// TIA Portal V17 export
// export: Created 2023-04-03T06:31:28.7566362Z, ExportSetting WithDefaults, DisplayName Totally Integrated Automation Portal, DisplayVersion V17 Update 4, DisplayName TIA Portal Openness, DisplayVersion V17 Update 4, DisplayName TIA Portal Version Control Interface, DisplayVersion V17, DisplayName STEP 7 Professional, DisplayVersion V17 Update 4, DisplayName STEP 7 Safety, DisplayVersion V17, DisplayName WinCC Professional, DisplayVersion V17 Update 4
FUNCTION "PN Com Read" : Void   // FC11, LAD
TITLE = ProfiNet Data Core <-> PEMS
{ S7_Optimized_Access := 'TRUE' }
VERSION : 0.1
// stored: AutoNumber false, IsIECCheckEnabled false, SetENOAutomatically false, UDAEnableTagReadback false
BEGIN

REGION Network 1: Read & Write Data From PEMS
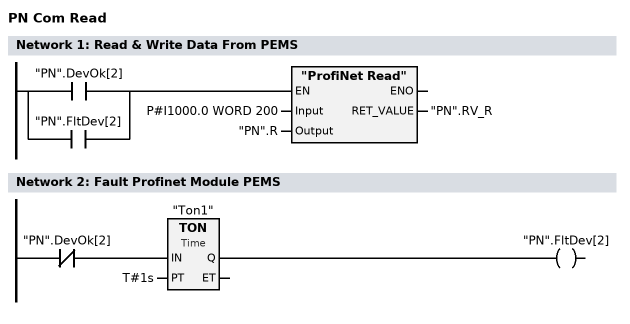
   RUNG wire#powerrail
      Contact( "PN".DevOk[2] )
      wire#w1
      "ProfiNet Read"(Input := P#I1000.0 WORD 200, Output := "PN".R, RET_VALUE => "PN".RV_R)
   END_RUNG
   RUNG wire#powerrail
      Contact( "PN".FltDev[2] )
   END_RUNG wire#w1
   // the same network as SCL:
   IF "PN".DevOk[2] OR "PN".FltDev[2] THEN
       "ProfiNet Read"(Input := P#I1000.0 WORD 200, Output := "PN".R, RET_VALUE => "PN".RV_R);
   END_IF;
END_REGION

REGION Network 2: Fault Profinet Module PEMS
   RUNG wire#powerrail
      I_Contact( "PN".DevOk[2] )
      { S7_Templates := "time_type := Time" } "Ton1".TON(pt := T#1s, et =>)
      Coil( "PN".FltDev[2] )
   END_RUNG
   // the same network as SCL:
   "Ton1".TON(IN := NOT "PN".DevOk[2], PT := T#1s);
   "PN".FltDev[2] := "Ton1".Q;
END_REGION
END_FUNCTION
